{attribute 'GeneratedUsingTerminal: EK1100-0000-0018'}
{attribute addProperty BoxType "EK1100-0000-0018"}
{attribute addProperty Id "Beckhoff_EKM1xxxEK1122Beckhoff_EKM1xxxEK1122_F03648A5412"}
{attribute addProperty CRC "609256685"}
{attribute addProperty Size "412"}
TYPE Beckhoff_EKM1xxx_245084ED EXTENDS EK1100_1FC0878B :
STRUCT
	{attribute addProperty Name "Beckhoff EKM1xxxEK1122"}
	{attribute addProperty PreviousPort "Beckhoff EKM1xxx : B"}
	Beckhoff_EKM1xxxEK1122 : Beckhoff_EKM1xxxEK1122_F03648A5;
END_STRUCT
END_TYPE

(* stored: Version 1.2.0.0, ProductVersion 3.1.4024.9
   DUT Beckhoff_EKM1xxx_245084ED: Id {32c60e75-f439-46a1-9d40-ccb91bc7882c} *)
